// Represents the current parsing state and is passed along
// as the parsing proceeds.
// All the public methods are intended to be invoked only by the generated code,
// users should never invoke them directly.
{attribute 'no_explicit_call' := 'do not call this POU directly'} 
FUNCTION_BLOCK FINAL FB_ParseContext
VAR_INPUT
END_VAR
VAR_OUTPUT
END_VAR
VAR
    stCtx   : ST_ParseContext;
END_VAR

VAR
END_VAR

// Internal-only property; when set to true, unknown fields will be discarded while parsing.
PROPERTY INTERNAL DiscardUnknownFields : BOOL
GET
DiscardUnknownFields := stCtx.stState.bDiscardUnknownFields;
END_GET
SET
stCtx.stState.bDiscardUnknownFields := DiscardUnknownFields;
END_SET
END_PROPERTY

METHOD FromBuffer : HRESULT
VAR_IN_OUT CONSTANT
    aBuffer : ARRAY [*] OF BYTE;
END_VAR

Reset();
Initialize(F_SpanFromArray(aBuffer));
END_METHOD

METHOD INTERNAL Initialize
VAR_INPUT CONSTANT
    stBuffer    : ST_Span;    
END_VAR
stCtx.stBuffer := stBuffer;

stCtx.stState.nBufferSize       := stBuffer.nSize;
stCtx.stState.nSizeLimit        := Param_PB.cMaxProtobufRawBuffer;
stCtx.stState.nRecursionLimit   := Param_PB.cRecursionLimit; 
stCtx.stState.nCurrentLimit     := TO_UDINT(-1);

stCtx.pCurrentContext 			:= THIS;
END_METHOD

// Initialize a ST_ParseContext using existing ST_ParserInternalState,
METHOD INTERNAL InitializeFromState
VAR_IN_OUT CONSTANT
    stState : ST_ParserInternalState;
    stBuffer : ST_Span;    
END_VAR
THIS^.stCtx.stState  := stState;
THIS^.stCtx.stBuffer := stBuffer;

stCtx.pCurrentContext := THIS;
END_METHOD

// Returns the last tag read, OR 0 IF no tags have been read OR we've read beyond the end of the input.
PROPERTY INTERNAL LastTag : UDINT
GET
LastTag := stCtx.stState.nLastTag;
END_GET
END_PROPERTY

METHOD ReadBool : HRESULT
VAR_OUTPUT
    bValue : BOOL;
END_VAR
VAR
    nTmp : BYTE;
END_VAR

ReadBool := F_ParseRawVarint32(THIS^.stCtx, nTmp);
bValue := nTmp <> 0;
END_METHOD

METHOD ReadBytes : HRESULT
VAR_IN_OUT
    aBytes : ARRAY [*] OF BYTE;
END_VAR
VAR_OUTPUT
	nCount : UDINT;
END_VAR

ReadBytes := F_ReadBytes(THIS^.stCtx, aBytes, nLength=> nCount);
END_METHOD

METHOD PUBLIC ReadDouble : HRESULT
VAR_OUTPUT
    fValue : LREAL;
END_VAR

ReadDouble := F_ParseDouble(THIS^.stCtx, fValue=> fValue);
END_METHOD

METHOD PUBLIC ReadEnum : HRESULT
VAR_INPUT
    anyEnum : ANY;
END_VAR
VAR
    nTmp   : UDINT;
	nCopySize : UDINT;
	retVal : UDINT;
END_VAR
IF anyEnum.pValue = NULL OR anyEnum.TypeClass <> __SYSTEM.TYPE_CLASS.TYPE_ENUM THEN
	ReadEnum := E_HRESULTAdsErr.INVALIDDATA;
	RETURN;
END_IF

ReadEnum := F_ParseRawVarint32(THIS^.stCtx, nTmp);
IF FAILED(ReadEnum) THEN
	RETURN;
END_IF

nCopySize := MIN(TO_UDINT(anyEnum.diSize), SIZEOF(nTmp));
IF nCopySize = 0 THEN
	ReadEnum := E_HRESULTAdsErr.INVALIDDATA;
	RETURN;
END_IF

MEMSET(destAddr:= anyEnum.pValue, fillByte:= 16#0, n:= TO_UDINT(anyEnum.diSize));
retVal := MEMCPY(destAddr:= anyEnum.pValue, srcAddr:= ADR(nTmp), n:= nCopySize);
IF retVal = 0 THEN
	ReadEnum := E_HRESULTAdsErr.INVALIDDATA;
END_IF
END_METHOD

METHOD PUBLIC ReadFixed32 : HRESULT
VAR_OUTPUT
    nValue : UDINT;
END_VAR

ReadFixed32 := F_ParseRawLittleEndian32(THIS^.stCtx, nValue=> nValue);
END_METHOD

METHOD PUBLIC ReadFixed64 : HRESULT
VAR_OUTPUT
    nValue : ULINT;
END_VAR

ReadFixed64 := F_ParseRawLittleEndian64(THIS^.stCtx, nValue=> nValue);
END_METHOD

METHOD PUBLIC ReadFloat : HRESULT
VAR_OUTPUT
    fValue : REAL;
END_VAR

ReadFloat := F_ParseFloat(THIS^.stCtx, fValue=> fValue);
END_METHOD

METHOD PUBLIC ReadInt32 : HRESULT
VAR_INPUT
    anyDint : ANY;
END_VAR
VAR
    nTmp   : UDINT;
	retVal : UDINT;
END_VAR

ReadInt32 := F_ParseRawVarint32(THIS^.stCtx, nTmp);
retVal := memcpy(destAddr:= anyDint.pValue, srcAddr:= ADR(nTmp), n:= MIN(TO_UDINT(anyDint.diSize), SIZEOF(nTmp)));
IF retVal = 0 THEN
	ReadInt32:= E_HRESULTAdsErr.INVALIDDATA;
END_IF
END_METHOD

METHOD PUBLIC ReadInt64 : HRESULT
VAR_INPUT
    anyLint : ANY;
END_VAR
VAR
    nTmp   : ULINT;
	retVal : UDINT;
END_VAR

ReadInt64 := F_ParseRawVarint64(THIS^.stCtx, nTmp);
retVal := memcpy(destAddr:= anyLint.pValue, srcAddr:= ADR(nTmp), n:= MIN(TO_UDINT(anyLint.diSize), SIZEOF(nTmp)));
IF retVal = 0 THEN
	ReadInt64:= E_HRESULTAdsErr.INVALIDDATA;
END_IF
END_METHOD

// Reads a length for length-delimited data.
METHOD PUBLIC ReadLength : HRESULT
VAR_OUTPUT
    nLength : UDINT;
END_VAR
ReadLength := F_ParseLength(THIS^.stCtx, nLength=> nLength);
END_METHOD

METHOD ReadMessage : HRESULT
VAR_INPUT
    ipMessage : I_Message;
END_VAR

ReadMessage := F_ReadMessage(fbCtx:= THIS^, ipMessage);
END_METHOD

METHOD PUBLIC ReadSFixed32 : HRESULT
VAR_OUTPUT
    nValue : DINT;
END_VAR
VAR
    nTmp : UDINT;
END_VAR

ReadSFixed32 := F_ParseRawLittleEndian32(THIS^.stCtx, nValue=> nTmp);

nValue := TO_DINT(nTmp);
END_METHOD

METHOD PUBLIC ReadSFixed64 : HRESULT
VAR_OUTPUT
    nValue : LINT;
END_VAR
VAR
    nTmp : ULINT;
END_VAR

ReadSFixed64 := F_ParseRawLittleEndian64(THIS^.stCtx, nValue=> nTmp);

nValue := TO_LINT(nTmp);
END_METHOD

METHOD PUBLIC ReadSInt32 : HRESULT
VAR_INPUT
    anyDint : ANY;
END_VAR
VAR
    nTmp   : UDINT;
	nValue : DINT;
	retVal : UDINT;
END_VAR

ReadSInt32 := F_ParseRawVarint32(THIS^.stCtx, nTmp);
nValue := F_DecodeZigZag32(nTmp);
retVal := memcpy(destAddr:= anyDint.pValue, srcAddr:= ADR(nValue), n:= MIN(TO_UDINT(anyDint.diSize), SIZEOF(nValue)));
IF retVal = 0 THEN
	ReadSInt32:= E_HRESULTAdsErr.INVALIDDATA;
END_IF
END_METHOD

METHOD PUBLIC ReadSInt64 : HRESULT
VAR_INPUT
    anyLint : ANY;
END_VAR
VAR
    nTmp   : ULINT;
	nValue : LINT;
	retVal : UDINT;
END_VAR

ReadSInt64 := F_ParseRawVarint64(THIS^.stCtx, nTmp);
nValue := F_DecodeZigZag64(nTmp);
retVal := memcpy(destAddr:= anyLint.pValue, srcAddr:= ADR(nValue), n:= MIN(TO_UDINT(anyLint.diSize), SIZEOF(nValue)));
IF retVal = 0 THEN
	ReadSInt64:= E_HRESULTAdsErr.INVALIDDATA;
END_IF
END_METHOD

METHOD PUBLIC ReadString : HRESULT
VAR_INPUT
    anyStringOut : ANY_STRING;
END_VAR
ReadString := F_ReadString(THIS^.stCtx, F_ToAnyType(anyStringOut));
END_METHOD

// Peeks at the next field tag. this is like calling "ReadTag", but the
// tag is not consumed. (So a subsequent call to "ReadTag" will return the same value.)
METHOD PUBLIC ReadTag : HRESULT
VAR_OUTPUT
    nTag : UDINT;
END_VAR
ReadTag := F_ParseTag(THIS^.stCtx, nTag=>nTag);
END_METHOD

METHOD PUBLIC ReadUint32 : HRESULT
VAR_INPUT
    anyUdint : ANY;
END_VAR
VAR
    nTmp   : UDINT;
	retVal : UDINT;
END_VAR

ReadUint32 := F_ParseRawVarint32(THIS^.stCtx, nTmp);
retVal := memcpy(destAddr:= anyUdint.pValue, srcAddr:= ADR(nTmp), n:= MIN(TO_UDINT(anyUdint.diSize), SIZEOF(nTmp)));
IF retVal = 0 THEN
	ReadUint32:= E_HRESULTAdsErr.INVALIDDATA;
END_IF
END_METHOD

METHOD PUBLIC ReadUint64 : HRESULT
VAR_INPUT
    anyUlint : ANY;
END_VAR
VAR
    nTmp   : ULINT;
	retVal : UDINT;
END_VAR

ReadUint64 := F_ParseRawVarint64(THIS^.stCtx, nTmp);
retVal := memcpy(destAddr:= anyUlint.pValue, srcAddr:= ADR(nTmp), n:= MIN(TO_UDINT(anyUlint.diSize), SIZEOF(nTmp)));
IF retVal = 0 THEN
	ReadUint64:= E_HRESULTAdsErr.INVALIDDATA;
END_IF
END_METHOD

PROPERTY refCtx : REFERENCE TO ST_ParseContext
GET
refCtx REF= THIS^.stCtx ;
END_GET
END_PROPERTY

METHOD PRIVATE Reset
VAR_INPUT
END_VAR

stCtx.stState.bError := FALSE;
stCtx.stState.eParserErrorCode := S_OK;
stCtx.stState.nBufferPos := 0;
stCtx.stState.nBufferSize := 0;
END_METHOD

METHOD SkipLastField : HRESULT
VAR_INPUT
END_VAR

SkipLastField := F_SkipLastField(THIS^.stCtx);
END_METHOD

END_FUNCTION_BLOCK

(* stored: Version 1.1.0.1
   POU FB_ParseContext: Id {33cf395e-4bc8-49aa-8a39-65170818d8f4}, SpecialFunc None
   Property DiscardUnknownFields: Id {00d117ed-687f-4a05-9f93-1740fbb958c8}
   Get Get: Id {9c267ab0-f51f-42a4-ade8-8b337d9756af}
   Set Set: Id {c0dc5b8c-1073-496a-91a1-e4aa0e7e1a93}
   Method FromBuffer: Id {2b7c5563-5ff2-4519-b454-28877ecfba59}
   Method Initialize: Id {8119bb60-2785-42c8-b5db-cc0a8f260d85}
   Method InitializeFromState: Id {49b2fb6e-7981-495b-912c-6024e1028cf7}
   Property LastTag: Id {3a0beeb8-51d3-475f-9d08-06678302f68f}
   Get Get: Id {41bb4c08-8917-4c55-b248-6149997987a6}
   Method ReadBool: Id {89c29bb6-d513-4d2b-aacf-0b905a1ea349}
   Method ReadBytes: Id {c954d0b9-35f8-44a1-a5f6-e08a7c90b59b}
   Method ReadDouble: Id {8d396e64-f286-4fda-95f4-0e77be4101f8}
   Method ReadEnum: Id {94929d12-39b1-4d65-901a-08d5f4ed083c}
   Method ReadFixed32: Id {8472785f-a763-4cc4-aa20-d1a39159ff5f}
   Method ReadFixed64: Id {343a76a1-067d-48aa-84aa-d005060019f6}
   Method ReadFloat: Id {ae5be64d-ac38-4693-99a6-f461c30093eb}
   Method ReadInt32: Id {98149cf0-c874-466c-84a8-ded7ed12b5d2}
   Method ReadInt64: Id {71d759ea-e908-4166-9283-378861c10204}
   Method ReadLength: Id {f8a2dea4-a747-4ce3-8692-a5ef550f442b}
   Method ReadMessage: Id {aa96c290-bd09-4969-a913-2cb9a48010fc}
   Method ReadSFixed32: Id {9f45ed62-393c-45d5-9752-212dd3ee0e22}
   Method ReadSFixed64: Id {73371c15-afa3-4f4d-84fd-bc8a39a6bb3d}
   Method ReadSInt32: Id {c895a857-fb22-484a-9a4e-0db57eebb101}
   Method ReadSInt64: Id {ee9a35c1-3c2f-4206-8072-64dc56e43c72}
   Method ReadString: Id {246de880-705a-44ea-a922-9753670627e5}
   Method ReadTag: Id {6e59f247-ef7c-45e6-b2dc-64a50e97c070}
   Method ReadUint32: Id {0a5f59af-f75a-4d04-8959-1ec62b11e925}
   Method ReadUint64: Id {01b6070b-c07f-4367-85e7-1d9c2c63ec50}
   Property refCtx: Id {889a9bbf-4ef8-4348-a5eb-48336314fc4d}
   Get Get: Id {b466954c-9fd1-43dc-9cfb-4a456eaa45e1}
   Method Reset: Id {09f049fb-0b8a-47f1-bb43-77baa133b86c}
   Method SkipLastField: Id {3e46d1b1-25c1-40fa-87b3-41790dad8370} *)
